TYPE E_InterlockState :
(
	UNDEFINED,
	Unlocked,
	Locked,
	Error
)USINT;
END_TYPE

(* stored: Version 1.1.0.1, ProductVersion 3.1.4020.6
   DUT E_InterlockState: Id {85b02c39-971e-4279-b4e4-81633269d89e} *)
